{attribute addProperty BoxType "AMP8000-0000-0103-0103"}
{attribute addProperty Id "Ch_A_ControlwordAT %Q*UINT162"}
{attribute addProperty CRC "456798364"}
{attribute addProperty SizeInBites "16"}
{attribute addProperty SizeInBytes "2"}
TYPE Ch_A_AxisMain_Outputs_1B3A309C :
STRUCT
	{attribute addProperty Name "Ch_A_Controlword"}
	Ch_A_Controlword AT %Q* : UINT;
END_STRUCT
END_TYPE

(* stored: Version 1.2.0.0, ProductVersion 3.1.4024.9
   DUT Ch_A_AxisMain_Outputs_1B3A309C: Id {98afe383-6a4e-4ef3-8ca7-6e10f1a09153} *)
